{attribute addProperty BoxType "EL6201-0000-0017"}
{attribute addProperty Id "Slave_7A_DI0BIT10.12549Slave_7A_DI1BIT10.12550Slave_7A_DI2BIT10.12551Slave_7A_DI3BIT10.12552Slave_7B_DI0BIT10.12553Slave_7B_DI1BIT10.12554Slave_7B_DI2BIT10.12555Slave_7B_DI3BIT10.12556"}
{attribute addProperty CRC "1665882461"}
{attribute addProperty SizeInBites "8"}
{attribute addProperty SizeInBytes "1"}
TYPE Slave_7_Inputs_634B595D :
STRUCT
	{attribute addProperty Name "Slave_7A_DI0"}
	Slave_7A_DI0 : BIT;
	{attribute addProperty Name "Slave_7A_DI1"}
	Slave_7A_DI1 : BIT;
	{attribute addProperty Name "Slave_7A_DI2"}
	Slave_7A_DI2 : BIT;
	{attribute addProperty Name "Slave_7A_DI3"}
	Slave_7A_DI3 : BIT;
	{attribute addProperty Name "Slave_7B_DI0"}
	Slave_7B_DI0 : BIT;
	{attribute addProperty Name "Slave_7B_DI1"}
	Slave_7B_DI1 : BIT;
	{attribute addProperty Name "Slave_7B_DI2"}
	Slave_7B_DI2 : BIT;
	{attribute addProperty Name "Slave_7B_DI3"}
	Slave_7B_DI3 : BIT;
END_STRUCT
END_TYPE

(* stored: Version 1.2.0.0, ProductVersion 3.1.4024.9
   DUT Slave_7_Inputs_634B595D: Id {bdb413d3-dd98-42ca-862b-db4abdaa07c8} *)
